FUNCTION_BLOCK Merge_Skill_Request (* Basic FB with empty ECC *)
  (* Standard: 61499-2 *)
  (* Version 1.0, 2023-02-20, AK125171 *)
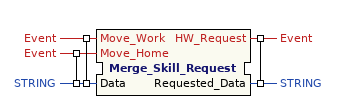
  EVENT_INPUT
    Move_Work WITH Data;
    Move_Home WITH Data;
  END_EVENT
  EVENT_OUTPUT
    HW_Request WITH Requested_Data;
  END_EVENT
  VAR_INPUT
    Data : STRING; (* WorkOrHome *)
  END_VAR
  VAR_OUTPUT
    Requested_Data : STRING;
  END_VAR
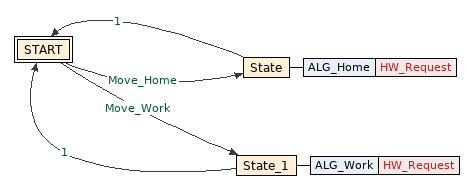
  EC_STATES
    START; (* Initial State *)
    State : ALG_Home -> HW_Request;
    State_1 : ALG_Work -> HW_Request;
  END_STATES
  EC_TRANSITIONS
    START TO State := Move_Home;
    START TO State_1 := Move_Work;
    State_1 TO START := 1;
    State TO START := 1;
  END_TRANSITIONS
  ALGORITHM ALG_Home IN ST:
Requested_Data:='Home';
  END_ALGORITHM
  ALGORITHM ALG_Work IN ST:
Requested_Data:='Work';
  END_ALGORITHM
END_FUNCTION_BLOCK
